Universal Robots PolyScope program: 7_wash_complete_to_hover.urp

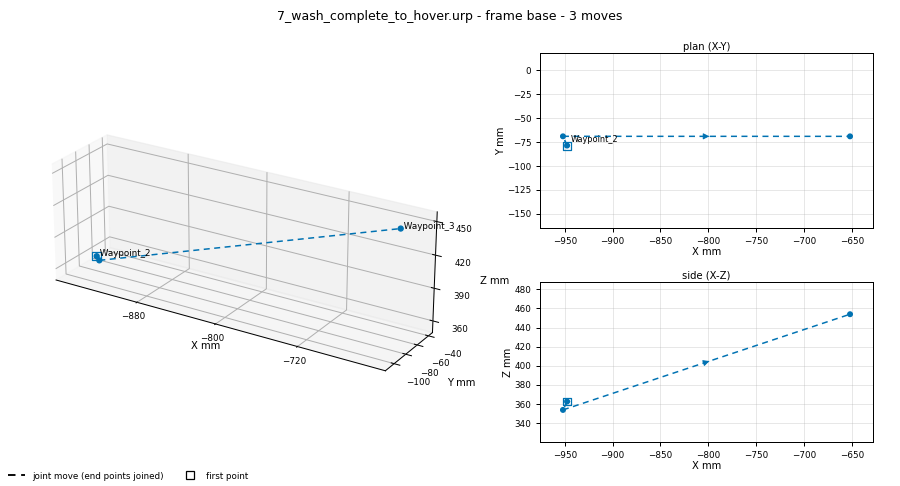
[picture p0: tool path of 7_wash_complete_to_hover.urp in frame base, 3 of 3 moves have a stored position in this frame; points joined in program order, loops and branches not executed]
Program 7_wash_complete_to_hover (installation=default directory=/programs/washer_rahman createdIn=5.9.5.1031259 lastSavedIn=5.9.5.1031259 robotSerialNumber=20215500597)
Calibrated DH parameters: a=[0.000193, -0.066673, -0.391568, -0.000012, 0.00005, 0]; d=[0.162643, -472.05677, 465.132521, 7.058239, 0.099746, 0.099582]; alpha=[1.571116, 0.00089, 0.003862, 1.569269, -1.569248, 0]; deltaTheta=[0, -1.413394, 7.628392, 0.068187, 0, -0.000001]
Robot Program (runOnlyOnce=true)
  MoveJ speed 60 deg/s, acceleration 80 deg/s^2 (useActiveTCP=true) feature=Base
    Waypoint Waypoint_2: TCP in base x=-947.576 y=-78.64 z=362.673 mm, rx=-1.3566 ry=-1.4371 rz=0.868 rad; joints [-2.083, -50.768, 70.998, -182.43, -94.111, -8.128] deg; TCP offset x=0 y=0 z=191.5 mm, rx=0 ry=0 rz=0 rad
    Waypoint Waypoint_1: TCP in base x=-951.865 y=-68.976 z=353.905 mm, rx=-1.3447 ry=-1.3257 rz=0.9789 rad; joints [-3.134, -48.014, 72.483, -192.566, -92.591, -4.137] deg
  MoveL speed 250 mm/s, acceleration 1200 mm/s^2 (useActiveTCP=true) feature=Base
    MoveDirectionNode (selectedDirection=ZPlus)
      Until DISTANCE (allowActions=false deceleration=3 distanceNodeType=STOP) Distance=0.1; motionParameters(blendRadius=0)
  MoveL speed 250 mm/s, acceleration 1200 mm/s^2 (useActiveTCP=true) feature=Base
    MoveDirectionNode (selectedDirection=XPlus)
      Until DISTANCE (allowActions=false deceleration=3 distanceNodeType=STOP) Distance=0.3; motionParameters(blendRadius=0)
  MoveJ speed 60 deg/s, acceleration 80 deg/s^2 (useActiveTCP=true) feature=Base
    Waypoint Waypoint_3: TCP in base x=-651.872 y=-69.005 z=453.916 mm, rx=-1.3447 ry=-1.3257 rz=0.9789 rad; joints [-5.79, -92.229, 118.135, -194.03, -90.03, -4.696] deg
